FUNCTION_BLOCK FB_MachineState EXTENDS FB_ListenerBase2
VAR_INPUT
	bCritical					:BOOL;				//クリティカルの発生
	bError						:BOOL;				//エラーの発生
	bWarning					:BOOL;				//ワーニングの発生
	bStay						:BOOL;				//McPowerがOFF
	bStop						:BOOL;				//McPowerがON
	bMoving						:BOOL;				//軸動作中または、（自動動作実行中（まだない））
END_VAR
VAR_OUTPUT
	eMachineState				:E_MachineState;	//マシーンステートを出力
	bStopMachine				:BOOL;				//モーションファンクションブロック停止
END_VAR
VAR
	fbListenerFilter			:FB_TcEventFilter;	//アラームフィルター

	liCriticalActiveCount		:LINT;				//クリティカル発生状況記憶
	liErrorActiveCount			:LINT;				//エラー発生状況記憶
	liWarningActiveCount		:LINT;				//ワーニング発生状況記憶
END_VAR

//---常に呼び出す必要があるので呼び出し---
	SUPER^.Execute();

//---発生アラームの重いほうからマシンステートに登録---
	IF bCritical=TRUE OR liCriticalActiveCount<>0 THEN
		eMachineState:=E_MachineState.Critical;
		bStopMachine:=TRUE;
		
	ELSIF bError=TRUE OR liErrorActiveCount<>0 THEN
		eMachineState:=E_MachineState.Error;
		bStopMachine:=TRUE;
	
	ELSIF bWarning=TRUE OR liWarningActiveCount<>0 THEN
		eMachineState:=E_MachineState.Warning;
		bStopMachine:=FALSE;
		
	ELSIF bStay=TRUE THEN
		eMachineState:=E_MachineState.Stay;
		bStopMachine:=FALSE;
		
	ELSIF bStop=TRUE THEN
		eMachineState:=E_MachineState.Stop;
		bStopMachine:=FALSE;
		
	ELSIF bMoving=TRUE THEN
		eMachineState:=E_MachineState.Moving;
		bStopMachine:=FALSE;
	END_IF

//FB_Init は常に暗黙的に使用可能で、主に初期化に使用されます。
//戻り値は評価されません。特定の結果を得るために、メソッドを明示的に宣言し、
//そのメソッドに標準の初期化コードをもったコードを追加することができます。戻り値を評価できます。
METHOD FB_Init: BOOL
VAR_INPUT
    bInitRetains: BOOL; // TRUE: 保持変数は初期化されます (ウォーム リセット、あるいはコールド リセット)
    bInCopyCode: BOOL;  // TRUE: 後でコードをコピーする (オンライン変更) ために、インスタンスをコピーします。
END_VAR
IF bInCopyCode = FALSE THEN
	
	//継承元のファンクションブロックの読み込むイベントのフィルター設定、アラームをフィルタリング
	fbListenerFilter.Clear().IsAlarm();
	
	//設定したフィルターを設定する
	SUPER^.Subscribe2(fbListenerFilter);

END_IF
END_METHOD

METHOD OnAlarmCleared : Tc3_EventLogger.HRESULT
VAR_INPUT
	fbEvent	: REFERENCE TO Tc3_EventLogger.FB_TcEvent;
END_VAR
CASE fbEvent.eSeverity OF 
	TcEventSeverity.Critical:
		liCriticalActiveCount:=liCriticalActiveCount-1;
		
	TcEventSeverity.Error:
		liErrorActiveCount:=liErrorActiveCount-1;
		
	TcEventSeverity.Warning:
		liWarningActiveCount:=liWarningActiveCount-1;
END_CASE

OnAlarmCleared:=S_OK;
END_METHOD

METHOD OnAlarmRaised : Tc3_EventLogger.HRESULT
VAR_INPUT
	fbEvent	: REFERENCE TO Tc3_EventLogger.FB_TcEvent;
END_VAR
CASE fbEvent.eSeverity OF 
	TcEventSeverity.Critical:
		liCriticalActiveCount:=liCriticalActiveCount+1;
		
	TcEventSeverity.Error:
		liErrorActiveCount:=liErrorActiveCount+1;
		
	TcEventSeverity.Warning:
		liWarningActiveCount:=liWarningActiveCount+1;
END_CASE

OnAlarmRaised:=S_OK;
END_METHOD

END_FUNCTION_BLOCK

(* stored: Version 1.1.0.1, ProductVersion 3.1.4026.18
   POU FB_MachineState: Id {c973bc40-a96e-4db3-9daa-2f59595f3f57}, SpecialFunc None
   Method FB_Init: Id {8e42fe74-f83c-423a-8ff8-6748f25ea1ea}
   Method OnAlarmCleared: Id {4dfafb76-ef14-4b92-a28e-252c1f7de862}
   Method OnAlarmRaised: Id {a6466c72-8d5a-419e-8150-cf5e66a31f3b} *)
